(* CoDeSys 2.3 export: CAPACITYBATCHERSUBSTATUS.EXP *)

(* Data type in ENUM *)
TYPE CapacityBatcherSubStatus : (CapacityBatcherSubStatusNormal:=0, CapacityBatcherSubStatusBatching, CapacityBatcherSubStatusPause,
										CapacityBatcherSubStatusRefStopped, CapacityBatcherSubStatusRefAlarm, CapacityBatcherSubStatusConfErr,
										CapacityBatcherSubStatusForbiddenCommand, CapacityBatcherSubStatusUnknownCommand, CapacityBatcherSubStatusBadCommandParameter);
END_TYPE
